{attribute 'GeneratedUsingTerminal: EP6224-0042-0016'}
{attribute addProperty BoxType "EP6224-0042-0016"}
{attribute addProperty Id "Module_1_DeviceState_Inputs_DeviceModule_1_DeviceState_Inputs_Device_5322301C2Module_2_DeviceState_InputsModule_2_DeviceState_Inputs_BD6C70354Module_7_Digital_InputsModule_7_Digital_Inputs_DAAE149B8WcStateAT %I*WcState_9091E0EB2InfoDataAT %I*InfoData_41C547A32"}
{attribute addProperty CRC "2959728762"}
{attribute addProperty Size "18"}
TYPE EP6224_B069E07A EXTENDS EtcSlaveTerminalBase_947E5A46 :
STRUCT
	{attribute addProperty Name "Module_1_DeviceState_Inputs_Device"}
	Module_1_DeviceState_Inputs_Device : Module_1_DeviceState_Inputs_Device_5322301C;
	{attribute addProperty Name "Module_2_DeviceState_Inputs"}
	Module_2_DeviceState_Inputs : Module_2_DeviceState_Inputs_BD6C7035;
	{attribute addProperty Name "Module_7_Digital_Inputs"}
	Module_7_Digital_Inputs : Module_7_Digital_Inputs_DAAE149B;
	{attribute addProperty Name "WcState"}
	WcState : WcState_9091E0EB;
	{attribute addProperty Name "InfoData"}
	InfoData : InfoData_41C547A3;
END_STRUCT
END_TYPE

(* stored: Version 1.2.0.0, ProductVersion 3.1.4024.9
   DUT EP6224_B069E07A: Id {03bdff42-d1ae-4ecd-9024-fca2b7add057} *)
